// TwinCAT 3 PLC project Untitled1
// Title: test1
// Company: blabla
// ProjectVersion: 0.0.1
// ProgramVersion: 3.1.4024.0
// project tree:
//   / MyLibFunction.TcPOU

// ---- MyLibFunction.TcPOU
FUNCTION_BLOCK MyLibFunction
VAR_INPUT
END_VAR
VAR_OUTPUT
END_VAR
VAR
END_VAR

END_FUNCTION_BLOCK
